// TIA Portal V17 export
// export: Created 2025-04-25T10:08:28.8098165Z, ExportSetting WithDefaults, DisplayName Totally Integrated Automation Portal, DisplayVersion V17 Update 8, DisplayName TIA Portal Openness, DisplayVersion V17 Update 8, DisplayName TIA Portal Version Control Interface, DisplayVersion V17, DisplayName SINAMICS Startdrive Advanced, DisplayVersion V17 SP2, DisplayName SINAMICS Startdrive G110M, G120, G120C, G120D, G120P, G115D, DisplayVersion V17 SP2, DisplayName SINAMICS Startdrive G130, G150, S120, S150, SINAMICS MV, S210, DisplayVersion V17 SP2, DisplayName STEP 7 Professional, DisplayVersion V17 Update 8, DisplayName SINUMERIK ONE STEP 7 Toolbox, DisplayVersion V17 Update 12, DisplayName SINUMERIK 840D sl STEP 7 Toolbox, DisplayVersion V17 Update 12, DisplayName STEP 7 Safety, DisplayVersion V17 Update 6, DisplayName WinCC Advanced / Unified PC, DisplayVersion V17 Update 8
DATA_BLOCK "DB22542_STIRRER_CONTROL_HOPPER_3_UNIT_2"   // DB22542
{ DB_Accessible_From_OPC_UA := 'FALSE' }
VERSION : 0.1
// stored: AutoNumber false, DBAccessibleFromOPCUA false, DBAccessibleFromWebserver true, InstanceOfName FB22502_STIRRER_CONTROL, InstanceOfType FB
"FB22502_STIRRER_CONTROL"
   // VAR_INPUT
   //    CONTROL_ON_DELAYED : Bool;
   //    MOTOR_CONDITIONS : Bool;
   //    MOTOR_STATUS_ERROR : Bool;
   //    MOTOR_STATUS_ENABLE : Bool;
   //    MOTOR_STATUS_REACHED : Bool;
   //    START_MANUAL_REQUEST : Bool;
   //    START_AUTO_REQUEST : Bool;
   //    START_PROGRAM_REQUEST : Bool;
   //    STOP_MANUAL_REQUEST : Bool;
   //    STOP_AUTO_REQUEST : Bool;
   //    STOP_PROGRAM_REQUEST : Bool;
   //    MOTOR_ACTUAL_POSITION : DInt;
   //    MOTOR_ACTUAL_VELOCITY : DInt;
   //    MOTOR_ACTUAL_CURRENT : DInt;
   //    MOTOR_ACTUAL_CURRENT_FILTERED : DInt;
   //    MOTOR_ACTUAL_TEMPERATURE : Real;
   //    MOTOR_STATUS_REGISTER : UDInt;
   // END_VAR
   // VAR_OUTPUT
   //    MOTOR_VELOCITY_TARGET_SOURCE : DInt;
   //    MOTOR_MODE_OF_OPERATION : Int;
   //    MOTOR_ENABLE_POWER_STAGE : Int;
   //    MOTOR_OUT1 : Bool;
   //    MOTOR_OUT2 : Bool;
   //    MOTOR_OUT3 : Bool;
   //    MOTOR_ENABLE_1 : Bool;
   //    MOTOR_ENABLE_2 : Bool;
   //    CURRENT_LIMIT_ALARM : Bool;
   //    TEMPERATURE_LIMIT_ALARM : Bool;
   // END_VAR
   // VAR
   //    DATA_STANDARD : "GENERAL_DATA_START_STOP";
   //    DATA_HMI : "HMI_DATA_START_STOP";
   //    INPUT_SETTINGS : Struct
   //       UNIT_NUMBER : Int := 2;
   //       HOPPER_NUMBER : Int := 3;
   //       MOTOR_REDUCTION : Int;
   //    END_STRUCT;
   //    ALARM_SETTINGS : Struct
   //       CURRENT_LIMIT : DInt;
   //       TEMPERATURE_LIMIT : Real;
   //       TIMER_CURRENT_LIMIT : TON_TIME;
   //       TIMER_TEMPERATURE_LIMIT : TON_TIME;
   //    END_STRUCT;
   //    HMI_MANUAL_SETPOINT_VELOCITY : DInt;
   //    HMI_ACTUAL_POSITION : DInt;
   //    HMI_ACTUAL_VELOCITY : DInt;
   //    HMI_ACTUAL_CURRENT : DInt;
   //    HMI_ACTUAL_CURRENT_FILTERED : DInt;
   //    HMI_STIRRER_LOW_RANGE : DInt;
   //    HMI_STIRRER_HIGH_RANGE : DInt;
   //    PROGRAM_SETPOINT_VELOCITY : DInt;
   //    SETPOINT_VELOCITY : DInt;
   //    FEEDBACK_POSITION : DInt;
   //    FEEDBACK_VELOCITY : DInt;
   //    FEEDBACK_CURRENT : DInt;
   //    FEEDBACK_CURRENT_FILTERED : DInt;
   //    FEEDBACK_TEMPERATURE : Real;
   //    HMI_PROGRAM_SETPOINT_VELOCITY : DInt;
   //    HMI_SETPOINT_VELOCITY : DInt;
   // END_VAR
BEGIN
END_DATA_BLOCK
